# EPICS alarm handler configuration: mps_database/bare/alarms/areas/mpln_spd_mp03.alhConfig
GROUP NULL MPLN:SPD:MP03:1
$ALIAS MPS Link Node 94
$GUIDANCE
LTUH MPS
   Group Name: MPLN:SPD:MP03:1
   Summary PV:  MPLN:SPD:MP03:1:STATSUMY
$END
CHANNEL  MPLN:SPD:MP03:1    MPLN:SPD:MP03:1:MPS_EN_RBV		-----
CHANNEL  MPLN:SPD:MP03:1    MPLN:SPD:MP03:1:LC1_MODE_RBV		-----
